// SIMATIC S7-200 project (STEP 7-Micro/WIN), CPU 222 REL 01.21

SYMBOL_TABLE USR1
SZ_A0            M0.0     // A0选择键
SZ_A1            M0.1     // A1选择键
SZ_A2            M0.2     // A2选择键
SZ_A3            M0.3     // A3选择键
SZ_A4            M0.4     // A4选择键
SZ_01            M0.5     // 预设尺寸1选择键
SZ_02            M0.6     // 预设尺寸2选择键
BL_SW            M1.0     // 底光开/关键
FL_SW            M1.1     // 侧光开/关键
LP_01            M1.2     // 预设灯光1选择键
LP_02            M1.3     // 预设灯光2选择键
U_State          M1.4     // 上行指示
D_State          M1.5     // 下行指示
SZ_AD            M2.0     // 尺寸增加键
SZ_RD            M2.1     // 尺寸减小键
SZ_SA0           M3.0     // A0存储键
SZ_SA1           M3.1     // A1存储键
SZ_SA2           M3.2     // A2存储键
SZ_SA3           M3.3     // A3存储键
SZ_SA4           M3.4     // A4存储键
SZ_S01           M3.5     // 预设尺寸1存储键
SZ_S02           M3.6     // 预设尺寸2存储键
BL_AD            M4.0     // 底光增加键
BL_RD            M4.1     // 底光减小键
FL_AD            M4.2     // 侧光增加键
FL_RD            M4.3     // 侧光减小键
LP_S01           M4.4     // 预设灯光1存储键
LP_S02           M4.5     // 预设灯光2存储键
SZ_OK            M5.0     // 更改底图尺寸预设值确认键
SZ_Cancel        M5.1     // 更改底图尺寸预设值取消键
LP_OK            M5.2     // 更改灯光预设值确认键
LP_Cancel        M5.3     // 更改灯光预设值取消键
Revert_OK        M5.4     // 载入出厂预设值确认键
W_TIP            M5.6     // 显示等待信息
RUN              M5.7     // 开机键
Reset_OK         M8.1     // 镜头复位
BL_OK            M8.3     // 底光开启延时
END_SYMBOL_TABLE

SYMBOL_TABLE USR2
BAR_WT           VW102    // 等待时间进度条
BAR_SZ           VW104    // 底图尺寸
BAR_BL           VW106    // 底光亮度
BAR_FL           VW108    // 侧光亮度
Pn               VD200    // 计数器当前值
H_BZ             VD204    // 抱闸最大允许误差上限
L_BZ             VD208    // 抱闸最大允许误差下限
H_JD             VD540    // 精度上限
L_JD             VD544    // 精度下限
YS_A0            VD500    // A0预设值
YS_A1            VD504    // A1预设值
YS_A2            VD508    // A2预设值
YS_A3            VD512    // A3预设值
YS_A4            VD516    // A4预设值
YS_01            VD520    // 底图尺寸预设值1
YS_02            VD524    // 底图尺寸预设值2
YS_BL1           VW528    // 底光预设值1
YS_FL1           VW530    // 侧光预设值1
YS_BL2           VW532    // 底光预设值2
YS_FL2           VW534    // 侧光预设值2
JINGDU           VD600    // 尺寸控制精度
BL_RP            VD604    // 底光补偿
OUT_A            I0.0     // 旋转编码器A相输出
OUT_B            I0.1     // 旋转编码器B相输出
EL_SW            I0.3     // 下限位开关
Z_FK             I0.4     // 正转反馈
F_FK             I0.5     // 反转反馈
KA1              Q0.0     // 正转输出
KA2              Q0.1     // 反转输出
KA3              Q0.2     // 低速
KM1              Q0.3     // 底光接触器
KM2              Q0.4     // 侧光接触器
BL_OUT           AQW0     // 底光控制
FL_OUT           AQW2     // 侧光控制
END_SYMBOL_TABLE

SYMBOL_TABLE USS 协议
USS_LOW_V        VD1000   // (DWORD)在此键入 USS协议符号的起始地址。
USS_HIGH_V       VD1004
USS_TIME_OUT     VW1008
USS_I_LINE       VW1010
USS_DAT_PTR0     VD1012
USS_ACT_DRV0     VD1016
USS_CUR_DRV0     VD1020
USS_P0           V1024.0
USS_REQ_SNT0     V1024.1
USS_RETRY_P0     VB1025
USS_ERR_CODE     VB1026
USS_CS_D0        VD1027
USS_CS_W0        VW1027
USS_CS_W2        VW1029
USS_CS_B0        VB1027
USS_CS_B1        VB1028
USS_POLL_BUF     VB1031
USS_XMT_0        VB1046
USS_XMT_ADR0     VB1049
USS_X_STWD       VD1056
USS_X_BCC        VB1060
USS_X_DW1        VD1047
USS_X_DW5        VD1051
USS_X_DW9        VD1055
USS_X_DB13       VB1059
USS_RCV_BUF0     VB1061
USS_R_STX        VB1062
USS_R_LGE        VB1063
USS_R_ADR        VB1064
USS_R_STWD       VD1071
USS_R_DW1        VD1062
USS_R_DW5        VD1066
USS_R_DW9        VD1070
USS_R_W13        VW1074
USS_STAT_TAB     VB1076
USS_ADR_P0       VB1396
END_SYMBOL_TABLE

ORGANIZATION_BLOCK 主:OB1
TITLE=【【【【此程序控制缩微机，涉及的物理设备包括缩微机镜头电机和灯光装置。系统通过镜头电机和灯光装置的精确控制，确保拍摄过程高效且图像质量可靠。】】】】
// 
// 程序设计注释：
// 系统通过镜头电机和灯光装置的精确控制，确保拍摄过程高效且图像质量可靠。操作员按下开机键后，镜头通过反转输出驱动向下移动，寻找由下限位开关检测的零位。在此过程中，等待时间进度条显示等待时间。若下限位开关未在10到100的时间范围内触发，系统会置位光电开关故障报警，并停止反转输出，以确保镜头移动可控。到达零位后，镜头复位完成标志置位，计数器当前值初始化为0，完成复位。
// 复位完成后，操作员可通过A0选择键到预设尺寸2选择键选择预设位置，程序自动调整镜头到目标位置。在自动模式下，若计数器当前值高于精度上限，启动反转输出下移。若计数器当前值低于精度下限，启动正转输出上移。镜头移动时，正转输出和反转输出按需独立运行，以保持方向明确。当计数器当前值超出允许范围时，系统置位抱闸失灵报警。报警触发后，系统停止移动，确保镜头位置稳定。手动模式下，操作员可按尺寸增加键或尺寸减小键直接调整高度。调整时，若接近下限位开关，系统通过反转输出保持镜头在安全范围内。调整完成后，结果显示在底图尺寸上。手动模式下，计数器当前值根据操作保持在0到56900之间，以确保镜头位置合理。新的位置可通过A0存储键到预设尺寸2存储键保存，并在按下更改底图尺寸预设值确认键后生效。若按更改底图尺寸预设值取消键，则放弃更改。
// 灯光方面，操作员通过底光开关键和侧光开关键控制底光接触器和侧光接触器的开关。使用底光增加键、底光减小键调整底光亮度。使用侧光增加键、侧光减小键调整侧光亮度。底光亮度和侧光亮度根据按键操作保持在0到100之间，以保护灯光设备。调整底光亮度和侧光亮度时，系统通过短暂延时确保操作稳定。调整后的亮度通过底光控制和侧光控制输出PWM信号实现。预设灯光值可通过预设灯光1选择键或预设灯光2选择键加载。预设灯光值由预设灯光1存储键和预设灯光2存储键保存，并按更改灯光预设值确认键确认。若按更改灯光预设值取消键，则取消更改。
// 系统持续监控设备状态。若正转输出或反转输出启动后，计数器当前值在一定时间内无变化，系统置位电机故障报警。报警触发后，系统停止电机运行，避免设备损坏。若计数器当前值达到56900，则触发上限位报警。报警触发后，停止镜头移动。任何报警触发时，系统关闭电机并提示操作员。待问题解决后，按报警复位键启动反转输出并置位复位标志，以恢复正常状态。复位完成后，镜头复位完成标志置位后，反转输出仅在必要时启动，以维持系统稳定。
BEGIN
Network 1 // 初始化
//  
// 网络注释
//  
// 
LD     SM0.1
R      SZ_A0:M0.0, 7
R      U_State:M1.4, 2
R      SZ_AD:M2.0, 2
R      SZ_SA0:M3.0, 8
R      BL_AD:M4.0, 7
R      SZ_OK:M5.0, 7
R      M6.0, 4
R      M7.0, 3
R      M8.0, 4
R      M9.0, 8
R      KA1:Q0.0, 5
MOVW   +0, BAR_WT:VW102
Network 2
LD     SM0.0
CALL   报警:SBR2
Network 3 // 按下“开机”，向下寻找零位
// 
// 
LDN    M8.0
A      RUN:M5.7
S      W_TIP:M5.6, 1
S      M8.0, 1
AN     EL_SW:I0.3
AN     KA1:Q0.0
S      KA2:Q0.1, 1
Network 4 // 显示等待时间进度条
// 
// 
LD     M8.0
AN     Reset_OK:M8.1
TON    T41, +10
A      T41
INCW   BAR_WT:VW102
R      T41, 1
Network 5 // 到达零位
// 
// 
LD     M8.0
A      EL_SW:I0.3
LPS
R      KA2:Q0.1, 1
MOVD   +0, SMD38
MOVB   16#F8, SMB37
HDEF   0, 9
HSC    0
MOVW   +100, BAR_WT:VW102
AN     Reset_OK:M8.1
ATCH   INT_0:INT0, 12
ENI
LPP
S      Reset_OK:M8.1, 2
Network 6 // 镜头高度显示
// 
// 
LD     Reset_OK:M8.1
MOVD   HC0, Pn:VD200
MOVD   VD536, H_BZ:VD204
+D     +1000, H_BZ:VD204
MOVD   VD536, L_BZ:VD208
-D     +1000, L_BZ:VD208
DTR    Pn:VD200, VD300
MOVR   VD300, VD304
/R     57000.0, VD304
MOVR   VD304, VD308
*R     852.0, VD308
TRUNC  VD308, VD312
DTI    VD312, VW316
MOVW   VW316, BAR_SZ:VW104
+I     +200, BAR_SZ:VW104
Network 7 // 镜头状态指示
// 
// 
LD     Reset_OK:M8.1
LPS
A      Z_FK:I0.4
=      U_State:M1.4
LRD
A      F_FK:I0.5
=      D_State:M1.5
LRD
CALL   底图尺寸控制:SBR0
LPP
CALL   灯光控制:SBR1
Network 8 // 底灯预热
// 
// 
LD     RUN:M5.7
LPS
A      BL_SW:M1.0
=      KM1:Q0.3
AN     M8.2
MOVW   +32000, BL_OUT:AQW0
TON    T42, +10
A      T42
S      BL_OK:M8.3, 1
LPP
LPS
A      FL_SW:M1.1
=      KM2:Q0.4
LPP
AN     BL_SW:M1.0
R      BL_OK:M8.3, 1
Network 9 // 载入出厂设定值
// 
// 
LD     Reset_OK:M8.1
A      Revert_OK:M5.4
R      SZ_A0:M0.0, 7
R      LP_S01:M4.4, 2
MOVD   +56900, YS_A0:VD500
MOVD   +38390, YS_A1:VD504
MOVD   +23600, YS_A2:VD508
MOVD   +13175, YS_A3:VD512
MOVD   +5810, YS_A4:VD516
MOVD   +0, YS_01:VD520
MOVD   +0, YS_02:VD524
MOVD   16#320032, VD528
MOVD   16#500050, VD532
R      Revert_OK:M5.4, 1
Network 10 // 自动赋初值
// 
// 
LD     SM0.0
LPS
LDD<   JINGDU:VD600, +200
OD>    JINGDU:VD600, +600
ALD
MOVD   +400, JINGDU:VD600
LPP
LDR>   BL_RP:VD604, 10.0
OR<    BL_RP:VD604, -10.0
ALD
MOVR   0.0, BL_RP:VD604
END_ORGANIZATION_BLOCK

SUBROUTINE_BLOCK 底图尺寸控制:SBR0
TITLE= 
// 子程序注释
// 按 F1 获得帮助及举例程序
//  
BEGIN
Network 1 // 旋转编码器记数范围0~56900
// 
// 
LD     SM0.0
LPS
AD<=   SMD42, +0
MOVD   +0, SMD42
LRD
AD>    SMD42, +56900
MOVD   +56900, SMD42
LRD
AD<=   Pn:VD200, +0
R      KA2:Q0.1, 1
LPP
AD>    Pn:VD200, +56900
R      KA1:Q0.0, 1
Network 2 // 选择A0~A4或两个预设值
// 
// 
LD     SM0.0
LPS
A      SZ_A0:M0.0
EU
MOVB   1, MB0
MOVD   YS_A0:VD500, VD536
LRD
A      SZ_A1:M0.1
EU
MOVB   2, MB0
MOVD   YS_A1:VD504, VD536
LRD
A      SZ_A2:M0.2
EU
MOVB   4, MB0
MOVD   YS_A2:VD508, VD536
LRD
A      SZ_A3:M0.3
EU
MOVB   8, MB0
MOVD   YS_A3:VD512, VD536
LRD
A      SZ_A4:M0.4
EU
MOVB   16, MB0
MOVD   YS_A4:VD516, VD536
LRD
A      SZ_01:M0.5
EU
MOVB   32, MB0
MOVD   YS_01:VD520, VD536
LRD
A      SZ_02:M0.6
EU
MOVB   64, MB0
MOVD   YS_02:VD524, VD536
LPP
MOVD   VD536, H_JD:VD540
+D     JINGDU:VD600, H_JD:VD540
MOVD   VD536, L_JD:VD544
-D     JINGDU:VD600, L_JD:VD544
Network 3 // 自动状态，尺寸当前值高于精度上限，镜头下行
// 
// 
LDB<>  MB0, 0
EU
AD>    Pn:VD200, H_JD:VD540
AB=    MB9, 0
AN     KA1:Q0.0
LPS
AN     KA2:Q0.1
S      KA2:Q0.1, 1
LRD
MOVD   H_JD:VD540, SMD42
LRD
MOVB   16#B0, SMB37
LRD
HDEF   0, 9
LRD
HSC    0
LPP
R      M8.2, 1
Network 4 // 自动状态，尺寸当前值低于精度下限，镜头上行
// 
// 
LDB<>  MB0, 0
EU
AD<    Pn:VD200, L_JD:VD544
AB=    MB9, 0
AN     KA2:Q0.1
LPS
AN     KA1:Q0.0
S      KA1:Q0.0, 1
LRD
MOVD   L_JD:VD544, SMD42
LRD
MOVB   16#B8, SMB37
LRD
HDEF   0, 9
LRD
HSC    0
LPP
R      M8.2, 1
Network 5 // 手动状态，按上移或下移按钮
// 
// 
LDB=   MB0, 0
LPS
AN     SZ_RD:M2.1
LPS
A      SZ_AD:M2.0
LPS
AD<    Pn:VD200, +56900
AN     KA2:Q0.1
S      KA1:Q0.0, 1
LPP
AD>=   Pn:VD200, +56900
R      KA1:Q0.0, 1
LPP
AN     SZ_AD:M2.0
R      KA1:Q0.0, 1
LPP
AN     SZ_AD:M2.0
LPS
A      SZ_RD:M2.1
AN     EL_SW:I0.3
AN     KA1:Q0.0
S      KA2:Q0.1, 1
LPP
AN     SZ_RD:M2.1
R      KA2:Q0.1, 1
Network 6 // 确认更改底图尺寸预设值
//  
// 网络注释
//  
// 
LD     SZ_OK:M5.0
LPS
A      SZ_SA0:M3.0
MOVD   Pn:VD200, YS_A0:VD500
LRD
A      SZ_SA1:M3.1
MOVD   Pn:VD200, YS_A1:VD504
LRD
A      SZ_SA2:M3.2
MOVD   Pn:VD200, YS_A2:VD508
LRD
A      SZ_SA3:M3.3
MOVD   Pn:VD200, YS_A3:VD512
LRD
A      SZ_SA4:M3.4
MOVD   Pn:VD200, YS_A4:VD516
LRD
A      SZ_S01:M3.5
MOVD   Pn:VD200, YS_01:VD520
LRD
A      SZ_S02:M3.6
MOVD   Pn:VD200, YS_02:VD524
LRD
R      SZ_SA0:M3.0, 7
LPP
R      SZ_OK:M5.0, 1
Network 7 // 取消更改底图尺寸预设值
// 
// 
LD     SZ_Cancel:M5.1
R      SZ_SA0:M3.0, 7
R      SZ_Cancel:M5.1, 1
END_SUBROUTINE_BLOCK

SUBROUTINE_BLOCK 灯光控制:SBR1
TITLE= 
// 子程序注释
// 按 F1 获得帮助及举例程序
//  
BEGIN
Network 1 // 灯光选择：预设1，预设2
// 
// 
LD     SM0.0
LPS
A      LP_01:M1.2
MOVD   VD528, VD106
LPP
A      LP_02:M1.3
MOVD   VD532, VD106
Network 2 // 按下底光增加按钮
// 
// 
LD     BL_SW:M1.0
A      BL_AD:M4.0
LPS
AN     M6.0
LPS
AW<    BAR_BL:VW106, +100
INCW   VW110
LPP
S      M6.0, 1
LPP
A      M6.0
TON    T45, +2
A      T45
R      M6.0, 1
R      T45, 1
Network 3 // 按下底光减小按钮
// 
// 
LD     BL_SW:M1.0
A      BL_RD:M4.1
LPS
AN     M6.1
LPS
AW>    BAR_BL:VW106, +0
DECW   VW110
LPP
S      M6.1, 1
LPP
A      M6.1
TON    T46, +2
A      T46
R      M6.1, 1
R      T46, 1
Network 4 // 底光亮度转换
// 
// 
LD     SM0.0
ITD    VW110, VD112
DTR    VD112, VD116
MOVR   BL_RP:VD604, VD608
+R     50.0, VD608
MOVR   100.0, VD612
-R     VD608, VD612
MOVR   VD612, VD616
/R     100.0, VD616
MOVR   VD116, VD120
*R     VD616, VD120
MOVR   VD120, VD124
+R     VD608, VD124
TRUNC  VD124, VD128
DTI    VD128, BAR_BL:VW106
Network 5 // 按下侧光增加按钮
// 
// 
LD     FL_SW:M1.1
A      FL_AD:M4.2
LPS
AN     M6.2
LPS
AW<    BAR_FL:VW108, +100
INCW   BAR_FL:VW108
LPP
S      M6.2, 1
LPP
A      M6.2
TON    T47, +3
A      T47
R      M6.2, 1
R      T47, 1
Network 6 // 按下侧光减小按钮
// 
// 
LD     FL_SW:M1.1
A      FL_RD:M4.3
LPS
AN     M6.3
LPS
AW>    BAR_FL:VW108, +0
DECW   BAR_FL:VW108
LPP
S      M6.3, 1
LPP
A      M6.3
TON    T48, +3
A      T48
R      M6.3, 1
R      T48, 1
Network 7 // 确认更改灯光预设值
//  
// 网络注释
//  
// 
LD     LP_OK:M5.2
LPS
A      LP_S01:M4.4
MOVD   VD106, VD528
LRD
A      LP_S02:M4.5
MOVD   VD106, VD532
LRD
R      LP_S01:M4.4, 2
LPP
R      LP_OK:M5.2, 1
Network 8 // 取消更改灯光预设值
// 
// 
LD     LP_Cancel:M5.3
R      LP_S01:M4.4, 2
R      LP_Cancel:M5.3, 1
Network 9 // 灯光控制输出
// 
// 
LD     SM0.0
LPS
ITD    BAR_BL:VW106, VD400
ITD    BAR_FL:VW108, VD404
DTR    VD400, VD408
DTR    VD404, VD412
MOVR   VD408, VD416
/R     100.0, VD416
MOVR   VD412, VD420
/R     100.0, VD420
MOVR   VD416, VD424
*R     32000.0, VD424
MOVR   VD420, VD428
*R     32000.0, VD428
TRUNC  VD424, VD436
TRUNC  VD428, VD440
DTI    VD436, VW444
DTI    VD440, VW446
A      M8.2
MOVW   VW444, BL_OUT:AQW0
LPP
MOVW   VW446, FL_OUT:AQW2
END_SUBROUTINE_BLOCK

SUBROUTINE_BLOCK 报警:SBR2
TITLE= 
// 子程序注释
// 按 F1 获得帮助及举例程序
//  
BEGIN
Network 1 // 光电开关故障
//  
// 网络注释
//  
// 
LDN    EL_SW:I0.3
LDN    Reset_OK:M8.1
AW>    BAR_WT:VW102, +10
AW<    BAR_WT:VW102, +100
LD     Reset_OK:M8.1
AD<    Pn:VD200, +0
OLD
ALD
S      M9.0, 1
Network 2 // 抱闸失灵
// 
// 
LDB<>  MB0, 0
A      M8.2
LDD>=  Pn:VD200, H_BZ:VD204
OD<=   Pn:VD200, L_BZ:VD208
ALD
S      M9.1, 1
Network 3 // 电机故障及上限位报警
// 
// 
LD     KA1:Q0.0
O      KA2:Q0.1
A      Reset_OK:M8.1
LPS
AN     M7.2
MOVD   Pn:VD200, VD700
S      M7.2, 1
LRD
TON    T43, +10
LPP
A      T43
LPS
AD=    Pn:VD200, VD700
LPS
AD<    Pn:VD200, +56900
S      M9.2, 1
LPP
AD>=   Pn:VD200, +56900
S      M9.3, 1
LPP
R      M7.2, 1
R      T43, 1
Network 4 // 有报警切换到报警窗口
// 
// 
LD     M9.0
EU
LD     M9.1
EU
OLD
LD     M9.2
EU
OLD
LD     M9.3
EU
OLD
S      M7.1, 1
R      KA1:Q0.0, 2
Network 5 // 按下报警复位键
// 
// 
LD     M7.0
LPS
A      M9.0
LPS
AN     EL_SW:I0.3
S      KA2:Q0.1, 1
LRD
A      EL_SW:I0.3
R      M9.0, 1
LPP
AN     KA2:Q0.1
R      M7.0, 1
LRD
LD     M9.1
O      M9.2
ALD
R      M9.1, 2
R      M7.0, 1
LPP
A      M9.3
AD<    Pn:VD200, +57000
R      M9.3, 1
R      M7.0, 1
END_SUBROUTINE_BLOCK

INTERRUPT_BLOCK INT_0:INT0
TITLE= 
// 中断程序注释
// 按 F1 获得帮助及举例程序
//  
// 
BEGIN
Network 1 // 网络题目 (单行)
//  
// 网络注释
//  
// 
LDB<>  MB0, 0
R      KA1:Q0.0, 2
S      M8.2, 1
END_INTERRUPT_BLOCK
